(* IEC 61131-3 sources: TESTS/OpenPCS, 3 files *)

(* ---- FbTask1.ST ---- *)
FUNCTION_BLOCK FbTask1
VAR_EXTERNAL

END_VAR

VAR_INPUT
Ts_ms :UDINT := 100;
Reset :BOOL  := FALSE;
END_VAR

VAR_OUTPUT
Blink:BOOL :=FALSE;
END_VAR

VAR
Timer1 :UDINT;
END_VAR
(*Blink meandr period 10000ms*)

IF ((Timer1 >= 10000) OR Reset) THEN
Timer1 := 0;
ELSE
Timer1 := Timer1 + Ts_ms;
END_IF;

IF (Timer1 <= 5000) THEN
Blink := TRUE;
ELSE
Blink := FALSE;
END_IF;

END_FUNCTION_BLOCK

(* ---- FbTs_ms.ST ---- *)
FUNCTION_BLOCK FbTs_ms
VAR_EXTERNAL

END_VAR

VAR_INPUT
RTC_in :DATE_AND_TIME;
Reset :BOOL  := FALSE;
END_VAR

VAR_OUTPUT
Ts_ms :UDINT := 0;
END_VAR

VAR
RTC_cur :DATE_AND_TIME;
RTC_prev :DATE_AND_TIME;
RTC_delta_time :TIME;
RTC_delta_dint :DINT;
END_VAR
(*PLC previous scan time ms*)
IF (Reset) THEN
RTC_cur := RTC_in;
RTC_prev := RTC_in;
ELSE
RTC_cur := RTC_in;
RTC_delta_time := RTC_cur - RTC_prev;
RTC_prev := RTC_cur;
RTC_delta_dint := TIME_TO_DINT(RTC_delta_time);

  (*Limit 0...1500ms*)
  IF ((RTC_delta_dint >= 0) AND (RTC_delta_dint <= 1500)) THEN
  Ts_ms := DINT_TO_UDINT(RTC_delta_dint);
  ELSE
  Ts_ms := 0;
  END_IF;

END_IF;

END_FUNCTION_BLOCK

(* ---- main.ST ---- *)
PROGRAM main
VAR_EXTERNAL

END_VAR

VAR_GLOBAL

END_VAR

VAR
Reset  :BOOL := TRUE; (*PLC First scan*)
DbTask1: FbTask1;
DbGetTaskInfo :GetTaskInfo;
DbTs_ms :FbTs_ms; (*PLC previous scan time ms*)
DbGETSYSTEMDATEANDTIME :GETSYSTEMDATEANDTIME;
END_VAR
(*
HELLO WORD BLINK PROJECT.
VA 25-06-2022
infoteam OpenPCS 7.1
https://www.ascontecnologic.com/product/openpcs/?lang=en
https://www.gcanbus.com/products/plc-con-ru/
https://github.com/DIYPLC/LibPlc
*)

DbGetTaskInfo();

DbGETSYSTEMDATEANDTIME();
DbTs_ms.RTC_in := DbGETSYSTEMDATEANDTIME.ODT;
DbTs_ms.Reset := Reset;
DbTs_ms();

DbTask1.Ts_ms := DbTs_ms.Ts_ms;
DbTask1.Reset := Reset;
DbTask1();

IF (Reset = TRUE) THEN
Reset := FALSE;
END_IF;

END_PROGRAM
